FUNCTION_BLOCK PUBLIC FB_LampSetDirectDALIAdapter EXTENDS FB_Lamp
VAR
	fbLampSetDirectDALI		: FB_LampSetDirectDALI;
END_VAR

// Reduces the control value by 5 in the range of 10 to 254.
METHOD PUBLIC DimDown
IF (fbLampSetDirectDALI.nLightLevel >= 38.1) THEN
	fbLampSetDirectDALI.SetLightLevel(TO_BYTE(fbLampSetDirectDALI.nLightLevel - 12.7));
END_IF
IF (_ipObserver <> 0) THEN
	_ipObserver.Update(fbLampSetDirectDALI.nLightLevel);
END_IF
END_METHOD

// Increments the control value by 5 in the range of 10 to 254.
METHOD PUBLIC DimUp
IF (fbLampSetDirectDALI.nLightLevel <= 241.3) THEN
	fbLampSetDirectDALI.SetLightLevel(TO_BYTE(TO_LREAL(fbLampSetDirectDALI.nLightLevel) + 12.7));
END_IF
IF (_ipObserver <> 0) THEN
	_ipObserver.Update(fbLampSetDirectDALI.nLightLevel);
END_IF
END_METHOD

METHOD FB_init : BOOL
VAR_INPUT
	bInitRetains : BOOL; // if TRUE, the retain variables are initialized (warm start / cold start)
	bInCopyCode : BOOL;  // if TRUE, the instance afterwards gets moved into the copy code (online change)
END_VAR
SUPER^._bIsDALIDevice := TRUE;
END_METHOD

// Sets the control value to 0.
METHOD PUBLIC Off
fbLampSetDirectDALI.SetLightLevel(0);
IF (_ipObserver <> 0) THEN
	_ipObserver.Update(fbLampSetDirectDALI.nLightLevel);
END_IF
END_METHOD

// Sets the control value to 254.
METHOD PUBLIC On
fbLampSetDirectDALI.SetLightLevel(254);
IF (_ipObserver <> 0) THEN
	_ipObserver.Update(fbLampSetDirectDALI.nLightLevel);
END_IF
END_METHOD

END_FUNCTION_BLOCK

(* stored: Version 1.1.0.1, ProductVersion 3.1.4024.11
   POU FB_LampSetDirectDALIAdapter: Id {06500677-1ca5-4f9c-bbca-0dcd0188c3d3}, SpecialFunc None
   Method DimDown: Id {7a075584-61ed-49e7-aa80-b192dd0ff064}
   Method DimUp: Id {85c48a51-31d1-4f15-b30f-dd92b0da00a7}
   Method FB_init: Id {c7dfbe5b-1192-4543-b513-6493e1286df9}
   Method Off: Id {3106f1b1-a466-4aaf-bf7c-b90c0d8b4c22}
   Method On: Id {2094a9c9-f771-43f7-aa2d-1a5adb3e0e4e} *)
